Staubli VAL3: page.pgx

public program page(string& menuname[], num index)
// set all the page in english IF
begin
  //
  //  PAGE
  //
  switch index
    //
  endSwitch
end
